{attribute addProperty BoxType "EK1122-0000-0018"}
{attribute addProperty Id "Beckhoff_ATH2xxxsub_EK1100EK1100_179A0949162A_0001_ATH2000_0250_0022A_0001_ATH2000_0250_0022_1D2C94B611214A_0002_ATH2000_0250_0023A_0002_ATH2000_0250_0023_006314D511214A_0003_ATH2000_0250_0024ATH2000_9506A48267284A_0004_ATH2040_0250_0022ATH2040_9506A48267284A_0005_ATH2040_0250_0023ATH2040_9506A48267284A_0006_ATH2040_0250_0024ATH2040_9506A48267284A_0007_ATH2050_0500_0022ATH2050_9506A48267284A_0008_ATH2050_0500_0023ATH2050_9506A48267284A_0009_ATH2050_0500_0024ATH2050_9506A48267284A_0010_ATH2050_0501_0022ATH2050_9506A48267284A_0011_ATH2050_0501_0023ATH2050_9506A48267284A_0012_ATH2050_0501_0024ATH2050_9506A48267284"}
{attribute addProperty CRC "1667402734"}
{attribute addProperty SizeInBites "6960"}
{attribute addProperty SizeInBytes "870"}
TYPE Beckhoff_ATH2xxxEK1122_63628BEE EXTENDS EK1122_179A0949 :
STRUCT
	{attribute addProperty Name "Beckhoff_ATH2xxxsub_EK1100"}
	Beckhoff_ATH2xxxsub_EK1100 : EK1100_179A0949;
	{attribute addProperty Name "A_0001_ATH2000_0250_0022"}
	A_0001_ATH2000_0250_0022 : A_0001_ATH2000_0250_0022_1D2C94B6;
	{attribute addProperty Name "A_0002_ATH2000_0250_0023"}
	A_0002_ATH2000_0250_0023 : A_0002_ATH2000_0250_0023_006314D5;
	{attribute addProperty Name "A_0003_ATH2000_0250_0024"}
	A_0003_ATH2000_0250_0024 : ATH2000_9506A482;
	{attribute addProperty Name "A_0004_ATH2040_0250_0022"}
	A_0004_ATH2040_0250_0022 : ATH2040_9506A482;
	{attribute addProperty Name "A_0005_ATH2040_0250_0023"}
	A_0005_ATH2040_0250_0023 : ATH2040_9506A482;
	{attribute addProperty Name "A_0006_ATH2040_0250_0024"}
	A_0006_ATH2040_0250_0024 : ATH2040_9506A482;
	{attribute addProperty Name "A_0007_ATH2050_0500_0022"}
	A_0007_ATH2050_0500_0022 : ATH2050_9506A482;
	{attribute addProperty Name "A_0008_ATH2050_0500_0023"}
	A_0008_ATH2050_0500_0023 : ATH2050_9506A482;
	{attribute addProperty Name "A_0009_ATH2050_0500_0024"}
	A_0009_ATH2050_0500_0024 : ATH2050_9506A482;
	{attribute addProperty Name "A_0010_ATH2050_0501_0022"}
	A_0010_ATH2050_0501_0022 : ATH2050_9506A482;
	{attribute addProperty Name "A_0011_ATH2050_0501_0023"}
	A_0011_ATH2050_0501_0023 : ATH2050_9506A482;
	{attribute addProperty Name "A_0012_ATH2050_0501_0024"}
	A_0012_ATH2050_0501_0024 : ATH2050_9506A482;
END_STRUCT
END_TYPE

(* stored: Version 1.2.0.0, ProductVersion 3.1.4024.9
   DUT Beckhoff_ATH2xxxEK1122_63628BEE: Id {3b7b8e4e-e7fe-47c9-9c4b-6d914f3d4442} *)
